TYPE MC_CAM_REF :
STRUCT
END_STRUCT
END_TYPE

(* stored: Version 1.1.0.1, ProductVersion 3.1.4024.12
   DUT MC_CAM_REF: Id {be0dc9a0-5c05-4434-bb8d-dbd68e448de4} *)
